DATA_BLOCK "ST10_DBInterface_Stopper"
{ S7_Optimized_Access := 'FALSE' }
VERSION : 0.1
NON_RETAIN
// ATTRIBUTES
// AUTO_NUMBER = False
// BLOCK_NUMBER = 2602
// END_ATTRIBUTES
   STRUCT
      Stopper : Array[1..50] of "UDT_StopperInterface";
   END_STRUCT;


BEGIN

END_DATA_BLOCK

